{attribute addProperty BoxType "EJ1957-0000-0017"}
{attribute addProperty Id "OutputsOutputs_32B9F5E1324"}
{attribute addProperty CRC "3096033232"}
{attribute addProperty SizeInBites "32"}
{attribute addProperty SizeInBytes "4"}
TYPE Module_2_FSOUT_B889B7D0 :
STRUCT
	{attribute addProperty Name "Outputs"}
	Outputs  : Outputs_32B9F5E1;
END_STRUCT
END_TYPE

(* stored: Version 1.2.0.0, ProductVersion 3.1.4024.9
   DUT Module_2_FSOUT_B889B7D0: Id {5b72ae29-b243-406e-9829-8322b9f6ea2b} *)
